FUNCTION_BLOCK FB_GasCounter IMPLEMENTS  I_ImpulseSensor
(*The impulse sensor counts impulses on the input devices. This can be used for gas counter, which trigger cyclic impulses every time a certain 
amount of gas has passed.
Example for a gas counter:
To calculate the total amount of consumed gas of the connected gas counter, firstly the counter at the start of the monitoring process is needed.
Then you can add the amount of gas that triggers the impulse of the gas counter (e.g. 0.1 m³) multiplied with nImpulse to get an approximation of
the current gas counter value*)
VAR
	fChpGasVtot: REAL:=67868.4; // Initial value of gas counter at start of monitoring
	fChpGasImp: REAL:=0.1; // Amount of gas, that triggers the impulse sensor
	nImpulse: UINT := 0; // Current number of registered Impulses
	fValue: REAL := fChpGasVtot; // Current value of gas counter
	nOn AT %I* : BIT; // Input signal of impulse sensor (if set from FALSE to TRUE, nImpulse increases by one)
	Counter: CTU; // Counter object
END_VAR

METHOD FB_init : BOOL
VAR_INPUT
	bInitRetains : BOOL; // if TRUE, the retain variables are initialized (warm start / cold start)
	bInCopyCode : BOOL;  // if TRUE, the instance afterwards gets moved into the copy code (online change)
	fChpGasVtotal: REAL:=67868.4; // Initial value of gas counter at start of monitoring
	fChpGasImpulse: REAL:=0.1; // Amount of gas, that triggers the impulse sensor
END_VAR
fChpGasVtot:=fChpGasVtotal;
fChpGasImp:=fChpGasImpulse;
END_METHOD

PROPERTY nImpulses : UINT
GET
nImpulses := THIS^.nImpulse;
END_GET
SET
 THIS^.nImpulse:=nImpulses;
END_SET
END_PROPERTY

METHOD Run: BOOL
Counter(CU:=nOn); // Count up (if nOn is set from FALSE to TRUE)
nImpulse:=WORD_TO_UINT(Counter.CV); // Write current counter value as UINT
fValue:=fCHPGasVtot+nImpulse*fChpGasImp;
END_METHOD

END_FUNCTION_BLOCK

(* stored: Version 1.1.0.1, ProductVersion 3.1.4024.6
   POU FB_GasCounter: Id {ef793c63-f1dd-458d-9982-db52cb00f461}, SpecialFunc None
   Method FB_init: Id {efac4151-a654-410d-bbcb-b1763c41bae0}
   Property nImpulses: Id {aed0d181-6136-497c-b4a5-ef6e47bc1a8b}
   Get Get: Id {1d5cdb7e-ceec-4cdb-a2f7-d5230eab1e9d}
   Set Set: Id {7f2494c9-cd10-45ca-a17f-91abf0336487}
   Method Run: Id {2f383681-bc32-4027-8750-5382c350814d} *)
